TYPE Es_CoordenadasCaballeteLadoA_ladoB :
STRUCT
	LadoA : Es_CoordenadasCaballeteLadoA ;
	LadoB : Es_CoordenadasCaballeteLadoB ;
END_STRUCT
END_TYPE

(* stored: Version 1.1.0.1, ProductVersion 3.1.4024.11
   DUT Es_CoordenadasCaballeteLadoA_ladoB: Id {4363d8da-bd39-481d-a655-a94509e55e13} *)
